{attribute 'linkalways'} 
{attribute 'no_explicit_call' := 'This FB is a CLASS and must be accessed using methods or properties'}
{attribute 'enable_dynamic_creation'}
FUNCTION_BLOCK ChunkedRequestSessionData EXTENDS Disposable IMPLEMENTS I_ChunkedRequestSessionData
VAR
	maximumChunkSizeInBytes : UDINT;
	totalReceivedChunks : UDINT;
	totalExpectedChunks : UDINT;
	pPayloadBuffer : POINTER TO STRING;
	payloadBufferSize : UDINT;
END_VAR

METHOD PRIVATE CreateBuffer
VAR_INPUT
	SizeInBytes : UDINT;
END_VAR
payloadBufferSize := SizeInBytes;
pPayloadBuffer := __NEW(BYTE, SizeInBytes);
memset(pPayloadBuffer, 0, SizeInBytes);
END_METHOD

METHOD PRIVATE DestroyBuffer
VAR_INPUT
END_VAR
IF pPayloadBuffer = 0 THEN
	RETURN;
END_IF

__DELETE(pPayloadBuffer);
pPayloadBuffer := 0;
END_METHOD

METHOD FB_exit : BOOL
VAR_INPUT
	bInCopyCode : BOOL; // if TRUE, the exit method is called for exiting an instance that is copied afterwards (online change).
END_VAR
IF bInCopyCode THEN
	RETURN;
END_IF

DestroyBuffer();
END_METHOD

METHOD FB_init : BOOL
VAR_INPUT
	bInitRetains : BOOL; // if TRUE, the retain variables are initialized (warm start / cold start)
	bInCopyCode : BOOL;  // if TRUE, the instance afterwards gets moved into the copy code (online change)
	ChunkSizeInBytes : UDINT;
	ChunkCount : UDINT;
END_VAR
maximumChunkSizeInBytes := ChunkSizeInBytes;
totalExpectedChunks := ChunkCount;
CreateBuffer(ChunkSizeInBytes * ChunkCount);
END_METHOD

PROPERTY PUBLIC IsComplete : BOOL
GET
IsComplete := totalReceivedChunks = totalExpectedChunks;
END_GET
END_PROPERTY

PROPERTY PUBLIC PayloadAddress : POINTER TO STRING
GET
PayloadAddress := pPayloadBuffer;
END_GET
END_PROPERTY

PROPERTY PUBLIC PayloadSizeInBytes : UDINT
GET
PayloadSizeInBytes := payloadBufferSize;
END_GET
END_PROPERTY

METHOD PUBLIC TryAddChunkedPayload : BOOL;
VAR_INPUT
	PayloadAddress : POINTER TO STRING;
	PayloadSize : DINT;
	ChunkSequence : DINT;
END_VAR
VAR
	offset : UDINT;
	pBufferChunkLocation : POINTER TO BYTE;
END_VAR
IF totalReceivedChunks >= totalExpectedChunks THEN
	RETURN;
END_IF

IF DINT_TO_UDINT(PayloadSize) > maximumChunkSizeInBytes THEN
	RETURN;
END_IF

IF ChunkSequence <= 0 THEN
	RETURN;
END_IF

concat2(pPayloadBuffer, PayloadAddress, pPayloadBuffer, payloadBufferSize);
totalReceivedChunks := totalReceivedChunks + 1;

TryAddChunkedPayload := TRUE;
END_METHOD

END_FUNCTION_BLOCK

(* stored: Version 1.1.0.1, ProductVersion 3.1.4024.12
   POU ChunkedRequestSessionData: Id {99b41408-4cca-4749-b5ea-cc34ac4e8cbd}, SpecialFunc None
   Folder Constructor: Id {b2f03932-c0a7-4fe4-a604-837598c04c83}
   Folder Destructor: Id {f84b601d-779e-4ad4-b195-11bc1f60e4e2}
   Folder Private: Id {e024060d-d35c-4597-95b4-0cff4bf92202}
   Method CreateBuffer: Id {ef5e76d1-6f88-4dbe-8c69-fe6d45ff059a}
   Method DestroyBuffer: Id {4ed70f4f-4840-48da-bbee-f1b2190add5c}
   Method FB_exit: Id {6a2ccd47-29e4-4a99-9715-482cec32f0a1}
   Method FB_init: Id {e2e04fb1-93b2-42bb-abe5-7ae8b8a95ff1}
   Property IsComplete: Id {7a441761-6d12-4608-8d81-b8e846f1b4fa}
   Get Get: Id {cf782de7-bdbb-4118-8082-e7735d8e9273}
   Property PayloadAddress: Id {35a25d9f-39dc-42e1-a305-0ce971a3b2fc}
   Get Get: Id {0142df66-2c76-4394-8960-ce277420641c}
   Property PayloadSizeInBytes: Id {dd39ffcf-b0eb-46b8-ae64-6b4e786014e3}
   Get Get: Id {74a77183-f16e-45d6-b585-93edc7b81455}
   Method TryAddChunkedPayload: Id {ad3d576d-bd11-4286-8b2d-751760ad4719} *)
